	FUNCTION_BLOCK FB 396
	TITLE =G296M AIR SHUT SLIDE KILN 2
	//COPYRIGHT:    (C) 2009  BUHLER AG, CH-9240 UZWIL, SWITZERLAND
	//
	//PRODUCT:      WinCoS_BIW01_09
	//
	//TITLE:        AIR SHUT SLIDE KILN 2
	//                Machine group control
	//                Maschinengruppensteuerung
	//
	//--------------------------------------------------------------------------------
	//
	//IDENT:        AUTHOR:             DEPT:                              DATE:
	//
	//P01_FB396.1.0 K.Renz              CSB41                              13.Jan.2010
	//             1st Release
	//
	//--------------------------------------------------------------------------------
	//
	//PURPOSE:
	//
	//MANUAL :
	//
	//RESTRICTIONS:
	//
	//--------------------------------------------------------------------------------
	AUTHOR  : KR
	FAMILY  : USW
	VERSION : 9.9


	VAR
	  Gr       : FB10;	//Standard interface to group
	  InOutValue1    : DINT; //Data for user
	  InOutValue2    : DINT; //Data for user
	  OutWayConflict : BOOL;	//Data for user
	  OutSelectionOk : BOOL;	//Data for user
	  CmdNewValue : BOOL;	//Data for user
	  CmdNewJob   : BOOL;	//Data for user
	  OutCodeOK   : BOOL;	//Data for user
	  InEndOfJob  : BOOL ;	//Data for user
	  staWayOk      : BOOL ;	//Data for user
	  EdgeStartRelease : BOOL ;	//Data for user
	  USW8  : BOOL;	//Data for user
	  USW9 : BOOL;	//Data for user
	  USW10: BOOL;	//Data for user
	  USW11: BOOL;	//Data for user
	  USW12: BOOL;	//Data for user
	  USW13: BOOL;	//Data for user
	  USW14: BOOL;	//Data for user
	  USW15: BOOL;	//Data for user
	     #A_3201_MXZ01 : FB13;   // VLS
	END_VAR
	VAR_TEMP
	   tmpEnable		: BOOL;
	   tmpFlag  		: BOOL;
	   tmpCmdNext		: BOOL;
	   tmpLocal  		: BOOL;
	   tmpAspOk  		: BOOL;
	   tmpHWStop 		: BOOL;
	   tmpInstanzDBNo       : INT ;
	END_VAR
	BEGIN
	NETWORK
	TITLE =
	NETWORK
	TITLE =Read command from group control
	//Parameter
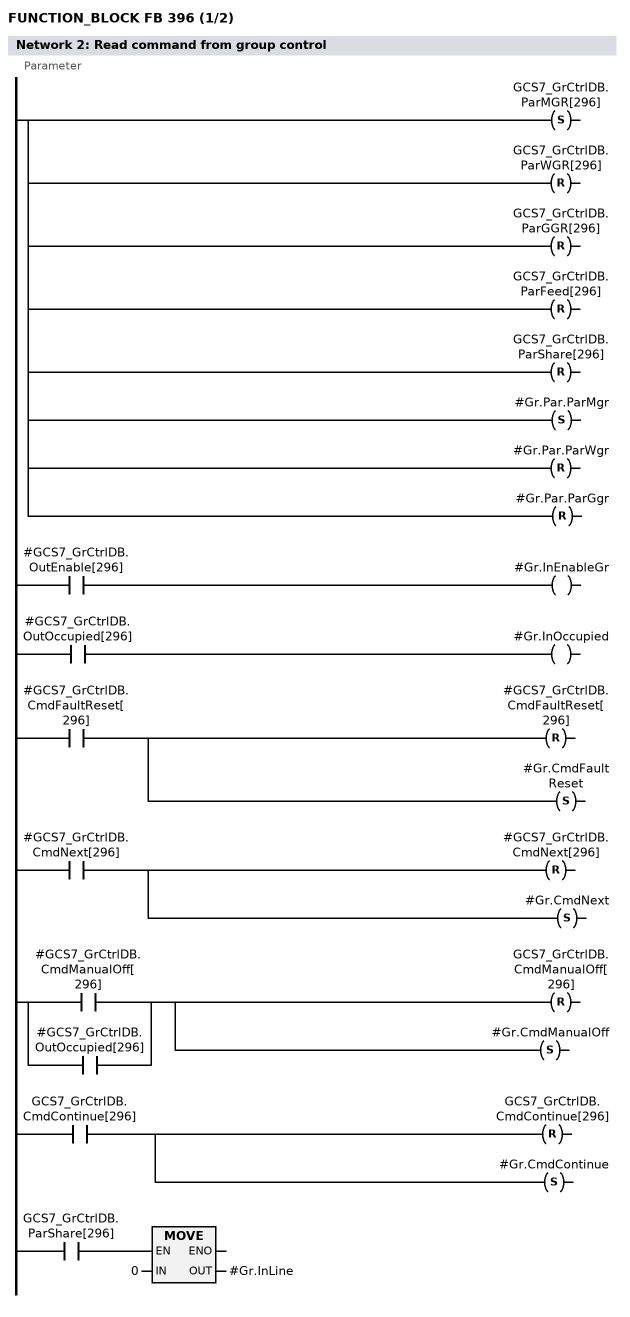
	      SET;
	      S   GCS7_GrCtrlDB.ParMGR[296];
	      R   GCS7_GrCtrlDB.ParWGR[296];
	      R   GCS7_GrCtrlDB.ParGGR[296];
	      R   GCS7_GrCtrlDB.ParFeed[296];
	      R   GCS7_GrCtrlDB.ParShare[296];
	      S   #Gr.Par.ParMgr;
	      R   #Gr.Par.ParWgr;
	      R   #Gr.Par.ParGgr;
	//Command
	      U   #GCS7_GrCtrlDB.OutEnable[296];
	      =   #Gr.InEnableGr;
	      U   #GCS7_GrCtrlDB.OutOccupied[296];
	      =   #Gr.InOccupied;
	      U   #GCS7_GrCtrlDB.CmdFaultReset[296];
	      R   #GCS7_GrCtrlDB.CmdFaultReset[296];
	      S   #Gr.CmdFaultReset;
	      U  #GCS7_GrCtrlDB.CmdNext[296];
	      R   #GCS7_GrCtrlDB.CmdNext[296];
	      S   #Gr.CmdNext;
	      U   #GCS7_GrCtrlDB.CmdManualOff[296];
	      O   #GCS7_GrCtrlDB.OutOccupied[296];
	      R   GCS7_GrCtrlDB.CmdManualOff[296];
	      S   #Gr.CmdManualOff;
	      U  GCS7_GrCtrlDB.CmdContinue[296];
	      R   GCS7_GrCtrlDB.CmdContinue[296];
	      S   #Gr.CmdContinue;
	//Init Line Number
	      U   GCS7_GrCtrlDB.ParShare[296];
	      SPBN WE00;
	      L     0;
	      T     #Gr.InLine;
	WE00: NOP   0;
	NETWORK
	TITLE =Call Methode Control
	// 1. Handle Interface PCControl
	// 2. Prepare mode --> ModePassive,ModeActive,ModeIdling
	// 3. Reset global flags of the group
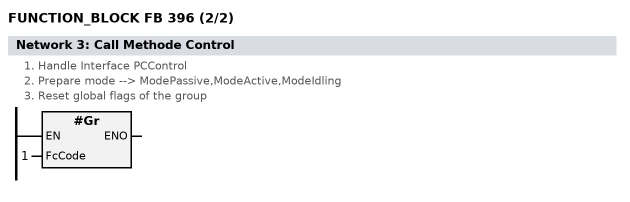
	      CALL #Gr (
	           FcCode                   := 1);
	NETWORK
	TITLE =Restart Idling Time
		L  #Gr.Par.ParIdling;
		L  2;
		>=I;
		SPB IdTm;
		T  #Gr.Par.ParIdling;
	IdTm:   NOP 0;
	      CLR;
	      S    #Gr.CmdRestartIdling;
	NETWORK
	TITLE =Prepare global flags
	NETWORK
	TITLE =Set Pattern (Target position)
	NETWORK
	TITLE =Interlocking WayOk
	//
	NETWORK
	TITLE =Interlocking Autostart
		CLR;
		R   #Gr.OutAutostart;
	NETWORK
	TITLE =Interlocking Enable
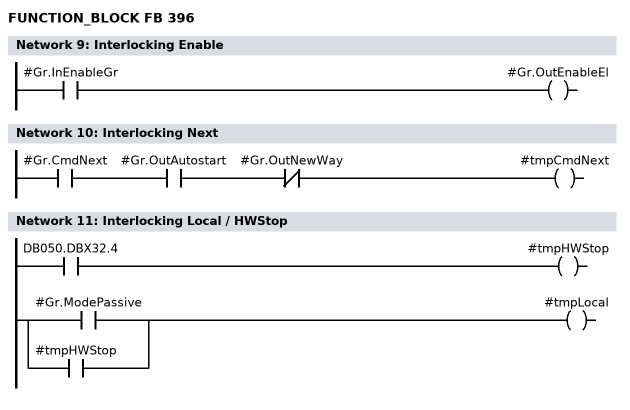
	      U     #Gr.InEnableGr;
	      =     #Gr.OutEnableEl;

	NETWORK
	TITLE =Interlocking Next
	      U     #Gr.CmdNext;
	      U     #Gr.OutAutostart;
	      UN    #Gr.OutNewWay;
	      =    #tmpCmdNext;

	NETWORK
	TITLE =Interlocking Local / HWStop
	      U    DB050.DBX32.4;
	      =    #tmpHWStop;

	      U    #Gr.ModePassive;
	      O    #tmpHWStop;
	      =    #tmpLocal;

	NETWORK
	TITLE ==A-3201-MXZ01 : OUTLET FLAP DRIVE
	NOP 0;
	//-InLocal---
	      U     #tmpLocal;
	      =     #A_3201_MXZ01.InLocal;
	//
	//-Interlocking---
	         =     #A_3201_MXZ01.InEnableHN;
	         NOT;
	         =     #A_3201_MXZ01.InEnableLN;
	//
	         SET;
	         S     #A_3201_MXZ01.CmdNext;
	//
	      U     #Gr.OutSeqStop;
	      =     #A_3201_MXZ01.InSeqStop;
	//
	//-Read inputs---
	      U     E 1008.0;
	      =     #A_3201_MXZ01.InpLN;
	      U     E 1008.1;
	      =     #A_3201_MXZ01.InpHN;
	      X     A 1004.0;
	      X     E 1004.0;
	      O;
	      X     A 1004.1;
	      X     E 1004.1;
	      =     #A_3201_MXZ01.InpFaultDev;
	      U   DB050.DBX32.4;
	      =     #A_3201_MXZ01.InHWStop;
	       U     PLC_DPInfo.Master[1].SlavesError[101];
	       =       #A_3201_MXZ01.InDPFault;
	//
	//-Set Parameters---
	//
	//-Call object control---
	      CALL  #A_3201_MXZ01;
	//
	//-Write outputs---
	      U     #A_3201_MXZ01.OutpLN;
	      =     A 1004.0;
	      U     #A_3201_MXZ01.OutpHN;
	      =     A 1004.1;
	NETWORK
	TITLE =Test Fault
	      U     #A_3201_MXZ01.StFault;
	      =     #Gr.VarFault;
	NETWORK
	TITLE =Test Warning
	      CLR;
	      =     #Gr.OutWarning;
	NETWORK
	TITLE =Test Stopped
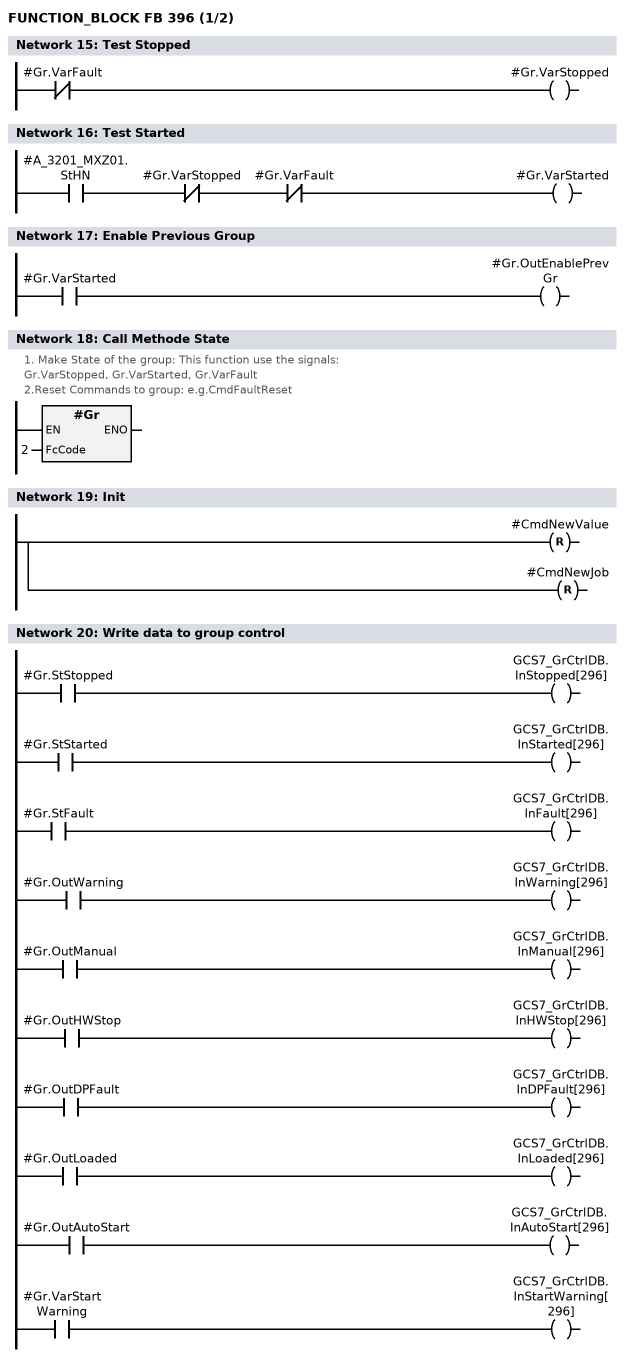
	      UN   #Gr.VarFault;
	      =     #Gr.VarStopped;
	NETWORK
	TITLE =Test Started
	      U     #A_3201_MXZ01.StHN;
	      UN  #Gr.VarStopped;
	      UN  #Gr.VarFault;
	      =     #Gr.VarStarted;
	NETWORK
	TITLE =Enable Previous Group
	      U    #Gr.VarStarted;
	      =     #Gr.OutEnablePrevGr;
	NETWORK
	TITLE =Call Methode State
	//1. Make State of the group: This function use the signals:
	//        Gr.VarStopped, Gr.VarStarted, Gr.VarFault
	//2.Reset Commands to group: e.g.CmdFaultReset
	      CALL #Gr (
	           FcCode                   := 2);
	NETWORK
	TITLE =Init
	      SET;
	      R    #CmdNewValue;
	      R    #CmdNewJob;
	NETWORK
	TITLE =Write data to group control
	      U   #Gr.StStopped;
	      =   GCS7_GrCtrlDB.InStopped[296];
	      U   #Gr.StStarted;
	      =   GCS7_GrCtrlDB.InStarted[296];
	      U   #Gr.StFault;
	      =   GCS7_GrCtrlDB.InFault[296];
	      U   #Gr.OutWarning;
	      =   GCS7_GrCtrlDB.InWarning[296];
	      U   #Gr.OutManual;
	      =   GCS7_GrCtrlDB.InManual[296];
	      U   #Gr.OutHWStop;
	      =   GCS7_GrCtrlDB.InHWStop[296];
	      U   #Gr.OutDPFault;
	      =   GCS7_GrCtrlDB.InDPFault[296];
	      U   #Gr.OutLoaded;
	      =   GCS7_GrCtrlDB.InLoaded[296];
	      U   #Gr.OutAutoStart;
	      =   GCS7_GrCtrlDB.InAutoStart[296];
	      U   #Gr.VarStartWarning;
	      =   GCS7_GrCtrlDB.InStartWarning[296];
	NETWORK
	TITLE =End of block
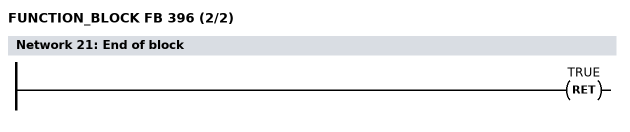

	BE

	END_FUNCTION_BLOCK
